// TIA Portal V16 export
// export: Created 2024-09-03T16:17:04.5561184Z, ExportSetting WithDefaults, DisplayName Totally Integrated Automation Portal, DisplayVersion V16, DisplayName TIA Portal Version Control Interface, DisplayVersion V16, DisplayName TIA Portal Openness, DisplayVersion V16, DisplayName STEP 7 Professional, DisplayVersion V16, DisplayName STEP 7 Safety, DisplayVersion V16, DisplayName WinCC Professional, DisplayVersion V16
ORGANIZATION_BLOCK "OB00001_IntINrmMainProgram"   // OB1, LAD, ProgramCycle
TITLE = Interrupt Module [NORMAL INTERRUPT] — Main Program Cyclic Execution
{ S7_Optimized_Access := 'TRUE' }
AUTHOR : M_Gledhill
FAMILY : Interrupt
NAME : IntINrmMainProgram
VERSION : 0.1
// PRACTICAL SERIES AUTOMATION LIBRARY (PAL)   —   COPYRIGHT 2020 – M. GLEDHILL (MIT LICENCE)
//                   ———— ◆ ————
// FULL ONLINE DOCUMENTATION IS AVAILABLE AT: https://practicalseries.com/2001-pal/index.html
// stored: AutoNumber true, IsIECCheckEnabled false, SetENOAutomatically false
   VAR_INPUT
      Initial_Call : Bool;   // Initial call of this OB
      Remanence : Bool;   // =True, if remanent data are available
   END_VAR
   VAR_TEMP
      revInfo : "UT01000_St_SysRevision";   // Revision information for this block
      licInfo : "UT01001_St_SysLicence";   // Licence information for this block
   END_VAR
BEGIN

REGION Network 1: Project description
   // ▄▄▄▄▄▄▄▄▄▄▄▄▄▄▄▄▄▄▄▄▄▄▄▄▄▄▄▄▄▄▄▄▄▄▄▄▄▄▄▄▄▄▄▄ 
   // 
   // 
   // TITLE:    PS2001 — PRACTICAL SERIES AUTOMATION LIBRARY
   // 
   // 
   // ▀▀▀▀▀▀▀▀▀▀▀▀▀▀▀▀▀▀▀▀▀▀▀▀▀▀▀▀▀▀▀▀▀▀▀▀▀▀▀▀▀▀▀▀ 
   // 
   // 
   // ――――――――――――――――――――――――――――――――――
   // COPYRIGHT:       © 2020 Michael Gledhill
   //           Part of the Practical Series of Publications
   //           Published in the United Kingdom
   //           mg@practicalseries.com
   //           https://practicalseries.com
   // ――――――――――――――――――――――――――――――――――
   // CUSTOMER:       Practical Series of Publications (PSP)
   // 
   // PROJECT:      Practical Series Automation Library (PAL)
   // 
   // PROJECT NO.:       PS2001
   // ――――――――――――――――――――――――――――――――――
   // CONTROLLER:       CPU 1515-2PN/DP
   // 
   // CONTROLLER NAME:    CON100
   // 
   // IP ADDRESS:      192.168.001.100
   // ――――――――――――――――――――――――――――――――――
   // TIA PROJECT NAME:    PS2001-PAL-D0018
   // STATUS:        DEVELOPMENT
   // ――――――――――――――――――――――――――――――――――
   // PROTECTION:     To minimise the risk of inadvertent modification to 
   //           tested modules, certain blocks will be released for 
   //           use with “protected access” (referred to a “write 
   //           protection” in Siemens terminology), this allows the 
   //           block to be used normally, but prevents the block 
   //           being accidentally modified. 
   // 
   //           This is in accordance with the risk assessment given 
   //           in the Validation Plant (VP), Appendix A [Ref. 002].
   // 
   //           ┌─────────────────────┐
   //           │ THE WRITE PROTECTION PASSWORD IS: PS2001 │
   //           └─────────────────────┘
   // 
   // 
   // ▄▄▄▄▄▄▄▄▄▄▄▄▄▄▄▄▄▄▄▄▄▄▄▄▄▄▄▄▄▄▄▄▄▄▄▄▄▄▄▄▄▄▄▄
   // PROJECT OVERVIEW
   // 
   // 
   // The PAL is a library of software modules and templates that have been developed for the 
   // Siemens Simatic S7-1500 range of controllers (and to a lesser extent the S7-1200 range).
   // 
   // The full library and all necessary documentation is available from the Practical Series website:
   // 
   //      https://practicalseries.com/2001-pal/index.html
   // 
   // 
   // The PAL is configured and deployed using the Siemens Simatic TIA Portal programming 
   // environment (version 16 or higher).
   // 
   // The PAL software structure is designed such that it is applicable to virtually all industrial 
   // applications that can generally controlled by a programmable logic controller.
   // 
   // The PAL software being developed as part of this Project, is considered to be suitable for use in 
   // the following types of industries (this is not an exhaustive list):
   // 
   //    •   Water and waste water treatment
   //    •   Pharmaceutical and batch production
   //    •   Brewing and fermentation
   //    •   Chemical manufacturing
   //    •   Oil and gas systems
   //    •   Food and beverage production
   // 
   // Such applications can generally be thought of as processes that operate with a response time
   // of more than 100 ms. I.e. the system would not be expected to respond to some stimuli faster
   // than 100 ms. In practice, a Controller may (and usually will) respond faster than this; however, 
   // a response time of 100 ms is considered to be an acceptable limit for PLC control.
   // 
   // At its most basic level, the PAL will be a library of software modules that control the fundamental 
   // aspects of an industrial plant; such modules would for example read the value of an instrument, 
   // operate a valve or drive, perform a calculation &c.
   // 
   // Such software modules are referred to as standard modules, these are fixed modules that 
   // perform a particular function and are identical across all software installations.
   // 
   // The PAL also contains application specific modules; these contain software that is applicable 
   // to the plant being controlled.
   // 
   // The Practical Series Automation Library is freely available under the MIT Open Source licence 
   // (see below). Those who find it useful may, if they wish, make a donation to support the library. 
   // 
   // Donations can be made here:
   // 
   //      https://practicalseries.com/2001-pal/11-web/81-00-pay.html
   // 
   // The PAL contains fully deployable software that has been developed by the author in his 
   // profession as a chartered electrical engineer. It is currently in use on various live plants 
   // throughout the UK and in some other parts of the world. 
   // 
   // This software is suitable for controlling and automating most industrial applications (typical 
   // process applications). It is easy to use and configure, but does have a degree of practical 
   // complexity appropriate for the environments within which it is employed. It is heavily 
   // configurable, has various operating modes and is suitable for a multitude of industrial 
   // applications.
   // 
   // IF YOU DON’T UNDERSTAND IT, DON’T USE IT. IF YOU DO USE IT, YOU DO SO AT YOUR OWN RISK.
   // 
   //                ━━━   ⬙⬙⬙⬙⬙⬙   ━━━
   // 
   // 
   // 
   // ▄▄▄▄▄▄▄▄▄▄▄▄▄▄▄▄▄▄▄▄▄▄▄▄▄▄▄▄▄▄▄▄▄▄▄▄▄▄▄▄▄▄▄▄
   // DOCUMENT REFERENCES
   // 
   //  ――――――――――――――――――――――――――――――――――――――――――
   //  REF.     DOCUMENT NO.       TITLE
   //  ――――――――――――――――――――――――――――――――――――――――――
   //  001  PS2001-5-0101-001   Quality Plan (QP)
   //  002  PS2001-5-0121-002   Validation Plan (VP)
   //  003  PS2001-5-0131-003   Test Plan (TP)
   //  004  PS2001-5-1101-001   User requirements specification (URS)
   //  005  PS2001-5-1111-001   Requirement Traceability Matrix (RTM)
   //  006  PS2001-5-2101-001   Functional Specification (FS) 
   //  007  PS2001-5-2211-001   Hardware Design Specification (HDS)
   //  008  PS2001-5-2311-001   Software Design Specification (SDS)
   //  009  PS2001-5-2313-011   Style Guide (SG)
   //  010  PS2001-5-234101-001    ES/WDP Configuration Manual
   //  011  PS2001-5-2312-fcNo.    Software Module Design Specification (SMDS)
   //  012  PS2001-5-2301-001   Software Module Register (SMR)
   //  013  PS2001-5-2302-011   Software Control and Mechanism (SCM)
   //  014  PS2001-5-7111-001   User Guide (UG)
   //  ――――――――――――――――――――――――――――――――――――――――――
   //  Note:   Where a block references another document not listed above (a calculation sheet
   //      for example), that document will be referenced separately in section 1.1 of the 
   //      block description for the block in question.
   // 
   // 
   // A full list of all project documentation is available here: 
   // 
   //      https://practicalseries.com/2001-pal/21-project/01-00-docs.html
   // 
   //                ━━━   ⬙⬙⬙⬙⬙⬙   ━━━
   // 
   // 
   // 
   // ▄▄▄▄▄▄▄▄▄▄▄▄▄▄▄▄▄▄▄▄▄▄▄▄▄▄▄▄▄▄▄▄▄▄▄▄▄▄▄▄▄▄▄▄
   // COMPLETED MODULES 
   // 
   //  ――――――――――――――――――――-―-- STATIC DATA       ― DYNAMIC  DAT A   ―
   //  BLOCK     NAME         REVISION    UDT/DB    REVISION  UDT/DB    REVISION  
   //  ――――――――――――――――――――――――――――――――――――――――――
   //  DB00801 St_ConstAiRawData  001.000   UT 00801   001.000       None
   //                  2024-05-16   DB00801   001.000       None
   //  ――――――――――――――――――――――――――――――――――――――――――
   //  DB00802 St_ConstAqRawData    001.000   UT 00802   001.000       None
   //                  2024-05-17   DB00802   001.000       None
   //  ――――――――――――――――――――――――――――――――――――――――――
   //  DB00851 St_ConstAiScaleData  001.000   UT 00851   001.000       None
   //                  2024-05-16   DB00851   001.000       None
   //  ――――――――――――――――――――――――――――――――――――――――――
   //  DB00851 St_ConstAqScaleData    001.000   UT 00852   001.000       None
   //                  2024-05-17   DB00852   001.000       None
   //  ――――――――――――――――――――――――――――――――――――――――――
   //  FC01001 StdSysGlobalData      002.000   None           UT 21000   002.000
   //                  2022-04-16                  UT 21001   002.000
   //                                    DB21001   002.000
   //  ――――――――――――――――――――――――――――――――――――――――――
   //  FC02001 StdInstAnalogRead    003.000   UT 02001   003.000    UT 22001   003.000
   //                  2024-05-16   DB02001   003.000       DB22001   003.000
   //  ――――――――――――――――――――――――――――――――――――――――――
   //  FC11001 StdDevValveIsol      002.000   UT 11001   002.000    UT 31001   002.000
   //                  2022-04-16   DB11001   002.000       DB31001   002.000
   //  ――――――――――――――――――――――――――――――――――――――――――
   //  FC11011 StdDevValve3Way      001.000   UT 11011   001.000    UT 31011   001.000
   //                  2022-06-11   DB11011   001.000       DB31011   001.000
   //  ――――――――――――――――――――――――――――――――――――――――――
   //  FC11101 StdDevValveBi      001.000   UT 11101   001.000    UT 31101   001.000
   //                  2023-02-02   DB11101   001.000       DB31101   001.000
   //  ――――――――――――――――――――――――――――――――――――――――――
   //  FC18001 StdSubScaleAI      003.000   None           None 
   //                  2022.08.31   None           None          
   //  ――――――――――――――――――――――――――――――――――――――――――
   //  FC18002 StdSubScaleAQ       001.000   None           None 
   //                  2022.09.01   None           None          
   //  ――――――――――――――――――――――――――――――――――――――――――
   //  FC18151 StdSubTimeEventRTC   002.000   None           UT 38151   002.000
   //                  2022-04-16   None           DB38151   002.000
   //  ――――――――――――――――――――――――――――――――――――――――――
   //  FC19511 StdDebugInst1Order    001.000   None           UT 39511   001.000
   //                  2023-03-03   None           DB39511   001.000
   //  ――――――――――――――――――――――――――――――――――――――――――
   //  FC19512 StdDebugInst2Order    002.000   None           UT 39512   002.000
   //                  2022-04-16   None           DB39512   002.000
   //  ――――――――――――――――――――――――――――――――――――――――――
   //  FC61000 DocGenExample     002.000   None           None 
   //                  2022-04-16   None           None          
   //  ――――――――――――――――――――――――――――――――――――――――――
   //  See Software Module Register [Ref. 012] for full details
   // 
   //                ━━━   ⬙⬙⬙⬙⬙⬙   ━━━
   // 
   // 
   // 
   // ▀▀▀▀▀▀▀▀▀▀▀▀▀▀▀▀▀▀▀▀▀▀▀▀▀▀▀▀▀▀▀▀▀▀▀▀▀▀▀▀▀▀▀▀
   // LICENCE AND CONTACT INFORMATION
   // 
   // This software and its associated documentation is made available under the MIT Licence:
   // 
   // ════════════════════════════════════════════
   // 
   // The MIT License (MIT)
   // 
   // Copyright © 2020 Michael Gledhill
   // 
   // Permission is hereby granted, free of charge, to any person obtaining a copy of this software 
   // and associated documentation files (the “Software”), to deal in the Software without restriction, 
   // including without limitation the rights to use, copy, modify, merge, publish, distribute, 
   // sublicense, and/or sell copies of the Software, and to permit persons to whom the Software is 
   // furnished to do so, subject to the following conditions: 
   // 
   // The above copyright notice and this permission notice shall be included in all copies or 
   // substantial portions of the Software.
   // 
   // THE SOFTWARE IS PROVIDED “AS IS”, WITHOUT WARRANTY OF ANY KIND, EXPRESS OR IMPLIED, 
   // INCLUDING BUT NOT LIMITED TO THE WARRANTIES OF MERCHANTABILITY, FITNESS FOR A 
   // PARTICULAR PURPOSE AND NON-INFRINGEMENT. IN NO EVENT SHALL THE AUTHORS OR COPYRIGHT 
   // HOLDERS BE LIABLE FOR ANY CLAIM, DAMAGES OR OTHER LIABILITY, WHETHER IN AN ACTION OF 
   // CONTRACT, TORT OR OTHERWISE, ARISING FROM, OUT OF OR IN CONNECTION WITH THE SOFTWARE 
   // OR THE USE OR OTHER DEALINGS IN THE SOFTWARE.
   // 
   // ════════════════════════════════════════════
   //                    ┌────────────┐
   // You can reach the author by email here:   │  mg@practicalseries.com  │
   //                    └────────────┘
   // Questions, corrections, constructive criticism and complaints (polite ones) are invited.
   // 
   // ▄▄▄▄▄▄▄▄▄▄▄▄▄▄▄▄▄▄▄▄▄▄▄▄▄▄▄▄▄▄▄▄▄▄▄▄▄▄▄▄▄▄▄▄
   // 
   //                ━━━   ⬙⬙⬙⬙⬙⬙   ━━━
   // 
   // 
   // 
   // ██████████████ █ █ █ █  END   █ █ █ █ ██████████████
END_REGION

REGION Network 2: Project revision and modification history
   // ▄▄▄▄▄▄▄▄▄▄▄▄▄▄▄▄▄▄▄▄▄▄▄▄▄▄▄▄▄▄▄▄▄▄▄▄▄▄▄▄▄▄▄▄
   // MODIFICATION HISTORY
   // 
   // The revision data herein contains the current revision of the whole software project 
   // (rather than of a particular block). The whole project is issued at a particular release and this is 
   // independent of individual module revisions.
   // 
   // The revision data shown here, in the network comments, contains additional information 
   // reflecting the software development workflow under the version control system (VCS) employed 
   // to track all software changes.
   // 
   // The VCS in use is the Git Source Code Management system in conjunction with the GitHub online 
   // hosting system. The software in its entirety is available in the GitHub remote repository:
   // 
   //      https://github.com/practicalseries/PS2001-pal-software
   // 
   // The repository is public and can be freely copied (forked in GitHub terminology) and used 
   // under the MIT licence. 
   // 
   // The MIT licence is reproduced in full in the last network of this software module.
   // 
   // 
   //  ———————————————————————————————————————————
   //  DATE       COMMIT TAG     AUTHOR        REASON FOR MODIFICATION
   //  ———————————————————————————————————————————
   //  2024.09.03    D0018      M. Gledhill      FC02001 — RELEASED FOR USE
   //                            FC18001 — RELEASED FOR USE
   //                            FC18002 — RELEASED FOR USE
   //                            DB00801, DB00802, DC00851 and
   //                            DB00852 all released for use
   // 
   //  2023.03.03    D0017      M. Gledhill      FC19511 — RELEASED FOR USE
   // 
   //  2023.02.02    D0016      M. Gledhill      FC11101 — RELEASED FOR USE
   // 
   //  2022.06.11    D0015      M. Gledhill      FC11011 — RELEASED FOR USE
   // 
   //  2022.05.03    D0014      M. Gledhill      Update to short URL links (now https)
   // 
   //  2022.04.16    D0011      M. Gledhill      All blocks — RE-RELEASED FOR USE
   //                            FC01001  FC02001  FC11001  FC18001 
   //                            FC18151  FC19152  FC61000
   // 
   //  2022.03.04    D0010      M. Gledhill      FC19512 — RELEASED FOR USE
   // 
   //  2021.08.23    D0009      M. Gledhill      FC11001 — RELEASED FOR USE
   // 
   //  2021.05.26    D0008      M. Gledhill      FC02001 — RELEASED FOR USE
   // 
   //  2021.05.22    D0007      M. Gledhill      FC18001 — RELEASED FOR USE
   // 
   //  2021.05.11    D0006      M. Gledhill      FC01001 — RELEASED FOR USE
   // 
   //  2021.05.02    D0005      M. Gledhill      Typographical corrections only
   // 
   //  2021.05.02    D0004      M. Gledhill      Typographical corrections only
   // 
   //  2021.02.19    D0003      M. Gledhill      FC18151 — RELEASED FOR USE
   // 
   //  2021.02.18    D0002      M. Gledhill      Baseline build
   // 
   //  2021.02.18    D0001      M. Gledhill      Hardware build
   // 
   //  2021.02.18    D0000      M. Gledhill      Initial commit — repository created
   //  ———————————————————————————————————————————
   // 
   // 
   // ▄▄▄▄▄▄▄▄▄▄▄▄▄▄▄▄▄▄▄▄▄▄▄▄▄▄▄▄▄▄▄▄▄▄▄▄▄▄▄▄▄▄▄▄
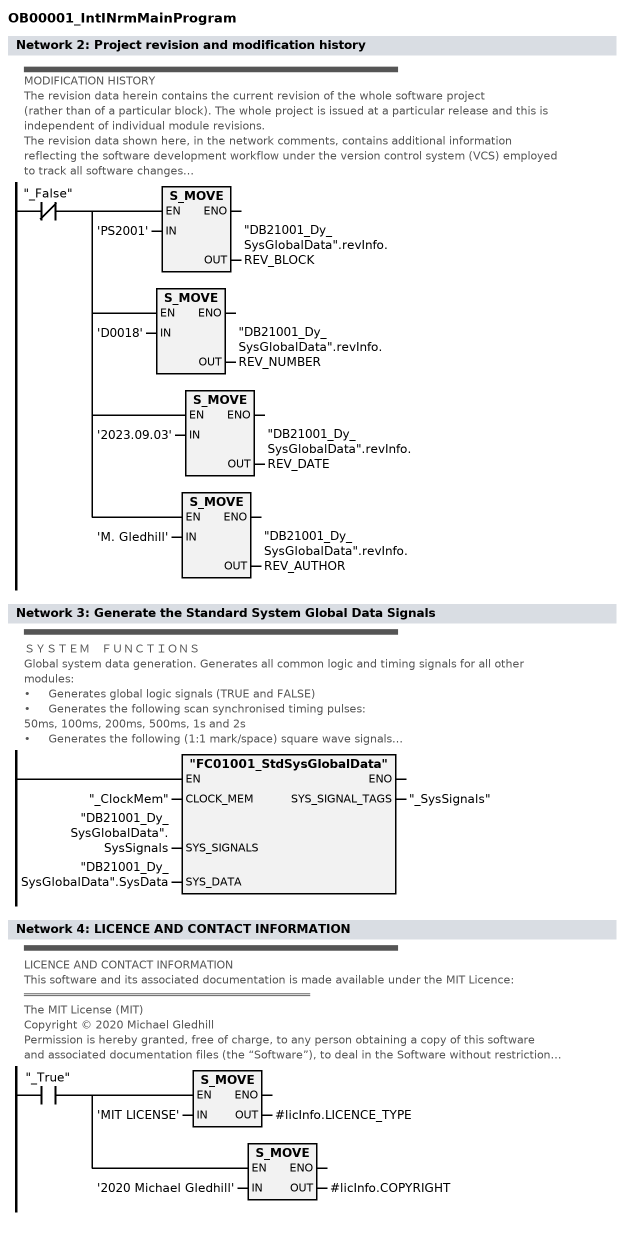
   RUNG wire#powerrail
      I_Contact( "_False" )
      wire#w1
      S_Move(in := 'PS2001', out => "DB21001_Dy_SysGlobalData".revInfo.REV_BLOCK)
   END_RUNG
   RUNG wire#w1
      S_Move(in := 'D0018', out => "DB21001_Dy_SysGlobalData".revInfo.REV_NUMBER)
   END_RUNG
   RUNG wire#w1
      S_Move(in := '2023.09.03', out => "DB21001_Dy_SysGlobalData".revInfo.REV_DATE)
   END_RUNG
   RUNG wire#w1
      S_Move(in := 'M. Gledhill', out => "DB21001_Dy_SysGlobalData".revInfo.REV_AUTHOR)
   END_RUNG
   // the same network as SCL:
   IF NOT "_False" THEN
       "DB21001_Dy_SysGlobalData".revInfo.REV_BLOCK := 'PS2001';
       "DB21001_Dy_SysGlobalData".revInfo.REV_NUMBER := 'D0018';
       "DB21001_Dy_SysGlobalData".revInfo.REV_DATE := '2023.09.03';
       "DB21001_Dy_SysGlobalData".revInfo.REV_AUTHOR := 'M. Gledhill';
   END_IF;
END_REGION

REGION Network 3: Generate the Standard System Global Data Signals
   // ▀▀▀▀▀▀▀▀▀▀▀▀▀▀▀▀▀▀▀▀▀▀▀▀▀▀▀▀▀▀▀▀▀▀▀▀▀▀▀▀▀▀▀▀
   // ＳＹＳＴＥＭ ＦＵＮＣＴＩＯＮＳ
   // 
   // Global system data generation. Generates all common logic and timing signals for all other 
   // modules:
   // 
   //    •   Generates global logic signals (TRUE and FALSE)
   // 
   //    •   Generates the following scan synchronised timing pulses:
   //        50ms, 100ms, 200ms, 500ms, 1s and 2s
   // 
   //    •   Generates the following (1:1 mark/space) square wave signals:
   //        100ms, 200ms, 500ms, 1s and 2s
   // 
   //    •   Generates odd and even (alternating) cycle tick-tock signals
   // 
   //    •   Generates a first-cycle signal indicating the controller has just started
   // 
   //    •   Records the cycle time of the last, maximum and minimum controller cycles
   // 
   //    •   Reads the controller internal real time clock and converts the values to discrete 
   //      integer values containing: year, month, day, day of week, hour, minute, second 
   //      and millisecond
   // 
   // The block must be the first non-debug block call within the main organisation block (OB 1).
   // ▄▄▄▄▄▄▄▄▄▄▄▄▄▄▄▄▄▄▄▄▄▄▄▄▄▄▄▄▄▄▄▄▄▄▄▄▄▄▄▄▄▄▄▄
   RUNG wire#powerrail
      "FC01001_StdSysGlobalData"(CLOCK_MEM := "_ClockMem", SYS_SIGNALS := "DB21001_Dy_SysGlobalData".SysSignals, SYS_DATA := "DB21001_Dy_SysGlobalData".SysData, SYS_SIGNAL_TAGS => "_SysSignals")
   END_RUNG
   // the same network as SCL:
   "FC01001_StdSysGlobalData"(CLOCK_MEM := "_ClockMem",
                           SYS_SIGNALS := "DB21001_Dy_SysGlobalData".SysSignals,
                           SYS_DATA := "DB21001_Dy_SysGlobalData".SysData,
                           SYS_SIGNAL_TAGS => "_SysSignals");
END_REGION

REGION Network 4: LICENCE AND CONTACT INFORMATION
   // ▀▀▀▀▀▀▀▀▀▀▀▀▀▀▀▀▀▀▀▀▀▀▀▀▀▀▀▀▀▀▀▀▀▀▀▀▀▀▀▀▀▀▀▀
   // LICENCE AND CONTACT INFORMATION
   // 
   // This software and its associated documentation is made available under the MIT Licence:
   // 
   // ════════════════════════════════════════════
   // 
   // The MIT License (MIT)
   // 
   // Copyright © 2020 Michael Gledhill
   // 
   // Permission is hereby granted, free of charge, to any person obtaining a copy of this software 
   // and associated documentation files (the “Software”), to deal in the Software without restriction, 
   // including without limitation the rights to use, copy, modify, merge, publish, distribute, 
   // sublicense, and/or sell copies of the Software, and to permit persons to whom the Software is 
   // furnished to do so, subject to the following conditions: 
   // 
   // The above copyright notice and this permission notice shall be included in all copies or 
   // substantial portions of the Software.
   // 
   // THE SOFTWARE IS PROVIDED “AS IS”, WITHOUT WARRANTY OF ANY KIND, EXPRESS OR IMPLIED, 
   // INCLUDING BUT NOT LIMITED TO THE WARRANTIES OF MERCHANTABILITY, FITNESS FOR A 
   // PARTICULAR PURPOSE AND NON-INFRINGEMENT. IN NO EVENT SHALL THE AUTHORS OR COPYRIGHT 
   // HOLDERS BE LIABLE FOR ANY CLAIM, DAMAGES OR OTHER LIABILITY, WHETHER IN AN ACTION OF 
   // CONTRACT, TORT OR OTHERWISE, ARISING FROM, OUT OF OR IN CONNECTION WITH THE SOFTWARE 
   // OR THE USE OR OTHER DEALINGS IN THE SOFTWARE.
   // 
   // ════════════════════════════════════════════
   //                    ┌────────────┐
   // You can reach the author by email here:   │  mg@practicalseries.com  │
   //                    └────────────┘
   // Questions, corrections, constructive criticism and complaints (polite ones) are invited.
   // 
   // ▄▄▄▄▄▄▄▄▄▄▄▄▄▄▄▄▄▄▄▄▄▄▄▄▄▄▄▄▄▄▄▄▄▄▄▄▄▄▄▄▄▄▄▄
   RUNG wire#powerrail
      Contact( "_True" )
      wire#w1
      S_Move(in := 'MIT LICENSE', out => #licInfo.LICENCE_TYPE)
   END_RUNG
   RUNG wire#w1
      S_Move(in := '2020 Michael Gledhill', out => #licInfo.COPYRIGHT)
   END_RUNG
   // the same network as SCL:
   IF "_True" THEN
       #licInfo.LICENCE_TYPE := 'MIT LICENSE';
       #licInfo.COPYRIGHT := '2020 Michael Gledhill';
   END_IF;
END_REGION
END_ORGANIZATION_BLOCK
